// Link between an input and an output group
FUNCTION_BLOCK FB_Link IMPLEMENTS I_Link
VAR
	IInputGroup				: I_DIGroup;				// Input group interface
	IOutputGroup			: I_DOGroup;				// Output group interface
	
	fbInputGroup			: FB_DIGroup;				// Input group FB, in case interface is not set to an FB
	fbOutputGroup			: FB_DOGroup;				// Output group FB, in case interface is not set to an FB
	
	stCommandTranslation	: ST_CommandTranslation;	// Input command to output command translation
	bExcludeFromOverview	: BOOL;						// Set to true to exclude this link from the links overview
END_VAR

// Get/set if the link needs to be excluded from the links overview
PROPERTY ExcludeFromOverview : BOOL
GET
ExcludeFromOverview := bExcludeFromOverview;
END_GET
SET
bExcludeFromOverview := ExcludeFromOverview;
END_SET
END_PROPERTY

// Pass the command from the input group to the output group
METHOD Execute
// Get input command and translate it to an output command
CASE IInputGroup.GetCommand() OF
	E_DICommand.None:
		IOutputGroup.SetCommand(E_DOCommand.None);
	E_DICommand.ShortPress:
		IOutputGroup.SetCommand(stCommandTranslation.OnShortPress);
	E_DICommand.DoublePress:
		IOutputGroup.SetCommand(stCommandTranslation.OnDoublePress);
	E_DICommand.LongPress:
		IOutputGroup.SetCommand(stCommandTranslation.OnLongPress);
	E_DICommand.Hold:
		IOutputGroup.SetCommand(stCommandTranslation.OnHold);
END_CASE

// Update output group indicators
IOutputGroup.DirectControl();

// Do not call the execute method of all IO groups here
// A digital in/output may appear in multiple links and the execute method should not be called more than once per PLC cycle
END_METHOD

METHOD FB_init : BOOL
VAR_INPUT
	bInitRetains : BOOL; // if TRUE, the retain variables are initialized (warm start / cold start)
	bInCopyCode : BOOL;  // if TRUE, the instance afterwards gets moved into the copy code (online change)
END_VAR
// Initialize interfaces with local FBs, can be replaced afterwards if needed
IInputGroup := fbInputGroup;
IOutputGroup := fbOutputGroup;
END_METHOD

// Group of inputs
PROPERTY InputGroup : I_DIGroup
GET
InputGroup := IInputGroup;
END_GET
SET
IInputGroup := InputGroup;
END_SET
END_PROPERTY

// Group of outputs
PROPERTY OutputGroup : I_DOGroup
GET
OutputGroup := IOutputGroup;
END_GET
SET
IOutputGroup := OutputGroup;
END_SET
END_PROPERTY

// Output reaction
PROPERTY OutputReaction : REFERENCE TO ST_CommandTranslation
GET
OutputReaction REF= stCommandTranslation;
END_GET
END_PROPERTY

END_FUNCTION_BLOCK

(* stored: Version 1.1.0.1, ProductVersion 3.1.4024.12
   POU FB_Link: Id {4bdfcc53-a26b-4e04-a8fa-6241c9f785b7}, SpecialFunc None
   Folder Methods: Id {57dd5418-cd8a-44ff-a950-1e53b6a2b33d}
   Folder Properties: Id {ef64cc13-6f9f-4c66-b9be-a6edd8f4c353}
   Property ExcludeFromOverview: Id {5cebf5de-44fa-407c-a7da-dcb80c71f22e}
   Get Get: Id {5d2869da-268e-48e5-9e2d-6c469d52bbc3}
   Set Set: Id {9986ab5d-e696-4175-911c-bba7029e00ad}
   Method Execute: Id {03b78132-bebc-4c43-b1d6-015f07efcbcd}
   Method FB_init: Id {68fa15b7-0a6f-454e-831e-4be7e69bf9b4}
   Property InputGroup: Id {b8e98866-4a22-4867-bd12-4fe6a4cb7d0e}
   Get Get: Id {7c2e7608-028d-48ad-94a1-d9d99e46c3ac}
   Set Set: Id {bcdcbcb5-d731-42aa-b712-c7f4db9644d5}
   Property OutputGroup: Id {72f6e40d-99e0-40f6-8cae-302d92986f9f}
   Get Get: Id {4c94efd2-d38e-4ccf-b66d-fbf6a63cb0ad}
   Set Set: Id {03aa02e5-5c62-4508-9440-48751e728753}
   Property OutputReaction: Id {871003ca-49ea-4200-9d92-ebff50c7ab04}
   Get Get: Id {63f201af-147f-4f6e-9765-0b687f0a4b91} *)
